FUNCTION_BLOCK LC_LED (* Composite Function Block Type *)
  (* Standard: 61499-2 *)
  (* Version 0.0, 2011-08-30, 4DIAC-IDE, 4DIAC-Consortium *)
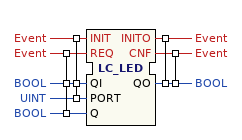
  EVENT_INPUT
    INIT WITH QI, PORT; (* Initialization Request *)
    REQ WITH QI, Q; (* Normal Execution Request *)
  END_EVENT
  EVENT_OUTPUT
    INITO WITH QO; (* Initialization Confirm *)
    CNF WITH QO; (* Execution Confirmation *)
  END_EVENT
  VAR_INPUT
    QI : BOOL; (* Input event qualifier *)
    PORT : UINT; (* Port # *)
    Q : BOOL; (* LED On/Off *)
  END_VAR
  VAR_OUTPUT
    QO : BOOL; (* Output event qualifier *)
  END_VAR
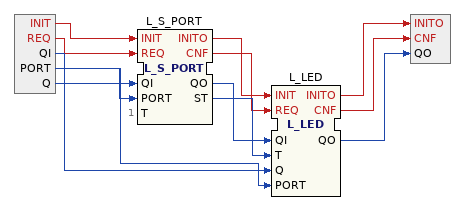
  FBS
    L_S_PORT : L_S_PORT(T := 1);
    L_LED : L_LED;
  END_FBS
  EVENT_CONNECTIONS
    INIT TO L_S_PORT.INIT;
    REQ TO L_S_PORT.REQ;
    L_S_PORT.INITO TO L_LED.INIT;
    L_S_PORT.CNF TO L_LED.REQ;
    L_LED.INITO TO INITO;
    L_LED.CNF TO CNF;
  END_CONNECTIONS
  DATA_CONNECTIONS
    QI TO L_S_PORT.QI;
    PORT TO L_S_PORT.PORT;
    L_S_PORT.QO TO L_LED.QI;
    L_S_PORT.ST TO L_LED.T;
    Q TO L_LED.Q;
    PORT TO L_LED.PORT;
    L_LED.QO TO QO;
  END_CONNECTIONS
END_FUNCTION_BLOCK
